PROGRAM MAIN
VAR
	fbAdder	:	FB_CalcAdder;
END_VAR

fbAdder(firstVar:= 5, secondVar:= 7, result=> );

END_PROGRAM

(* stored: Version 1.1.0.1, ProductVersion 3.1.4024.12
   POU MAIN: Id {39a59f10-14b9-4d6b-a642-f40e6fd55c02}, SpecialFunc None *)
